(* IEC 61131-3 sources: ProgettoAx_A_B/src, 3 files *)

(* ---- configuration.st ---- *)
USING Siemens.Simatic.S71500.Tasks;

CONFIGURATION Cfg
    TASK MyStartupTask : Startup;
    TASK MyProgramCycleTask : ProgramCycle;

    PROGRAM P1 WITH MyStartupTask : MyProgramStartup;
    PROGRAM P2 WITH MyProgramCycleTask : MyProgramMain;

        VAR_GLOBAL

            myOutput AT %Q0.0 : BOOL;
            myRealOutput AT %QW2 : INT;

        END_VAR

END_CONFIGURATION

(* ---- main.st ---- *)
PROGRAM MyProgramMain
    VAR_EXTERNAL
        //c : INT;
        //d : INT;
        //conflitto : BOOL;
        myRealOutput : INT;
    END_VAR

    VAR
    END_VAR

    myRealOutput := myRealOutput + 1;

END_PROGRAM

(* ---- startup.st ---- *)
PROGRAM MyProgramStartup
    VAR_EXTERNAL
        myOutput : BOOL;
    END_VAR

    myOutput := TRUE;

END_PROGRAM
